// TIA Portal V18 export
FUNCTION "TestBlock" : Void   // FC1, LAD
TITLE = What about this?
{ S7_Optimized_Access := 'TRUE' }
// stored: SetENOAutomatically false
   VAR_INPUT
      "Test input" : Bool;   // Hey!
   END_VAR
BEGIN

REGION Network 1: Other test comment
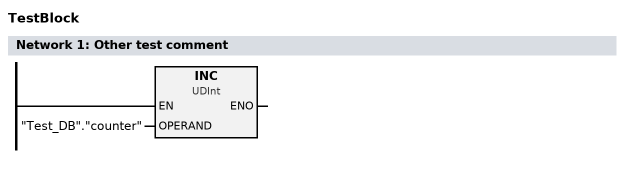
   RUNG wire#powerrail
      { S7_Templates := "DestType := UDInt" } Inc( "Test_DB"."counter" )
   END_RUNG
   // the same network as SCL:
   "Test_DB"."counter" := "Test_DB"."counter" + 1;
END_REGION
END_FUNCTION
